TYPE T_OCV_Filename : T_MaxString;
END_TYPE

(* stored: Version 1.1.0.1
   DUT T_OCV_Filename: Id {eceb38d8-0edd-4b0e-96eb-fc05333ffce3} *)
